Staubli VAL3: Main.pgx

program Main()
  local num l_nKey
begin
  //
  taskCreate "Move2P",10,MoveToPoint()

  do
    call Refresh()
    call RefreshList()
    call user:setList("点",sList,bUserRefresh,bListRefresh,nSelected,sItem,l_nKey)
    bUserRefresh=false
    bListRefresh=false
    call MainKey(l_nKey)
    delay(0)
  until bExit

end
